					GVL_MASTER.stNestTable.qNestRotatePortA := FALSE;
					GVL_MASTER.stNestTable.qNestRotatePortB := FALSE;
					GVL_MASTER.stNestTable.bNestInMotion    := FALSE;
				
					GVL_MASTER.stProcess.bNestTestingReady  := FALSE;
					GVL_MASTER.stProcess.bReleaseNestRotation := FALSE;
				
					GVL_MASTER.stNestTable.bSupportExtendRequest  := FALSE;
					GVL_MASTER.stNestTable.bSupportRetractRequest := TRUE;
				
					GVL_MASTER.stMachineStatus.eMachineState := E_MachineState.FAULT;

        END_CASE

    // =================================================================
    // FAULT 
    // =================================================================
	
	E_MachineState.FAULT:
	
	 				GVL_MASTER.stNestTable.qNestRotatePortA := FALSE;
					GVL_MASTER.stNestTable.qNestRotatePortB := FALSE;
					GVL_MASTER.stNestTable.bNestInMotion    := FALSE;
				
					GVL_MASTER.stProcess.bNestTestingReady  := FALSE;
					GVL_MASTER.stProcess.bReleaseNestRotation := FALSE;
				
					GVL_MASTER.stNestTable.bSupportExtendRequest  := FALSE;
					GVL_MASTER.stNestTable.bSupportRetractRequest := TRUE;

	    IF GVL_IO.stSafety.bSafetyOK AND NOT GVL_Master.stMachineStatus.bFault THEN
        	eNestState := E_NestState.IDLE;
        END_IF

	

		
	END_CASE
END_METHOD

METHOD PRIVATE M_OperatorExchangeControl
VAR
	iOperatorNestIndex 	: INT;
    bOperatorResultPass : BOOL;
    bOperatorResultFail : BOOL;
	bOperatorResultValid : BOOL;
END_VAR
// ============================================================================
// MERGED OPERATOR EXCHANGE CONTROL
//
// Base:
//     - Immediate retention of one-scan removal and reject pulses.
//     - Complete enabled/disabled Puck Locker behavior.
//     - Recovery if the Puck Locker mode changes during an exchange.
//
// Merge adjustments:
//     - Permit a pending PASS or FAIL result to be handled while another nest
//       is in TESTING.
//     - Prevent WaitingForPartLoading from blocking when the locker is disabled.
// ============================================================================
// Default value prevents stale index permission.
bOperatorExchangeComplete := FALSE;


// -----------------------------------------------------------------------------
// Validate the nest currently accessible to the operator.
// -----------------------------------------------------------------------------
IF eOperatorNestPosition = E_NestPosition.Unknown THEN
    RETURN;
END_IF


iOperatorNestIndex := TO_INT(eOperatorNestPosition);

IF (iOperatorNestIndex < 1) OR (iOperatorNestIndex > 4) THEN
    RETURN;
END_IF


// -----------------------------------------------------------------------------
// Result associated with the nest currently accessible to the operator.
// -----------------------------------------------------------------------------
bOperatorResultValid :=
    GVL_MASTER.astNestProcessResult[
        iOperatorNestIndex
    ].bResultValid;


bOperatorResultPass :=
    GVL_MASTER.astNestProcessResult[
        iOperatorNestIndex
    ].bResultValid
    AND
    GVL_MASTER.astNestProcessResult[
        iOperatorNestIndex
    ].bPass;


bOperatorResultFail :=
    GVL_MASTER.astNestProcessResult[
        iOperatorNestIndex
    ].bResultValid
    AND
    GVL_MASTER.astNestProcessResult[
        iOperatorNestIndex
    ].bFail;

// -----------------------------------------------------------------------------
// Retain operator actions even while the Kistler is processing another nest.
//
// Both the nest removal pulse and the reject sensor pulse last only one PLC
// scan. They must therefore be retained immediately and not only when the
// exchange state machine reaches the corresponding waiting state.
// -----------------------------------------------------------------------------

// A processed part was removed from the operator nest.
IF (
        bOperatorResultValid
        OR bPendingOperatorResultPass
        OR bPendingOperatorResultFail
   )
   AND GVL_MASTER.astNestTracking[
        iOperatorNestIndex
   ].bPartRemovedPulse THEN

    bPartRemovedConfirmedForExchange := TRUE;

END_IF


// -----------------------------------------------------------------------------
// A new part was loaded into the operator nest.
//
// The previous part result may remain latched in the exchange state machine,
// but the newly loaded physical part has not yet been tested.
//
// Clear only the HMI measurement/result so the new part is displayed as NONE.
// -----------------------------------------------------------------------------
IF GVL_MASTER.astNestTracking[
        iOperatorNestIndex
   ].bPartLoadedPulse THEN

    // Preserve the disposition of the removed part before clearing
    // the visual result for the newly loaded part.
    IF bOperatorResultValid THEN

        bPendingOperatorResultPass :=
            bOperatorResultPass;

        bPendingOperatorResultFail :=
            bOperatorResultFail;

    END_IF

    // The newly loaded part has not been tested yet.
    // Display NONE without losing the pending disposition above.
    M_HMIKistlerResult(
        eNestPosition := eOperatorNestPosition,
        bPartOK       := FALSE,
        bPartNOK      := FALSE,
        rForce        := 0.0,
        rDistance     := 0.0,
        bResetValues  := TRUE
    );

END_IF


// Reject confirmation is only valid after the failed part
// has been removed from the operator nest.
//
// Required order:
// 1. Remove the failed part from the nest.
// 2. Place the failed part at the reject sensor.
// 3. Complete the operator exchange.
IF (
        bOperatorResultFail
        OR bPendingOperatorResultFail
   )
   AND bPartRemovedConfirmedForExchange
   AND rtPartPresentReject.Q THEN

    bRejectConfirmedForExchange := TRUE;

END_IF


// ============================================================================
// Operator exchange sequence
// ============================================================================
CASE eOperatorExchangeState OF


    // ========================================================================
    E_OperatorExchangeState.Idle:
    // ========================================================================

        bOperatorExchangeComplete := FALSE;

        // Preserve the physical nest associated with this exchange.
        eCompletedOperatorExchangeNest :=
            eOperatorNestPosition;


        // --------------------------------------------------------------------
        // Case 1:
        // A tested result is pending at the operator nest.
        //
        // The processed part must be handled before the table may index.
        // --------------------------------------------------------------------
        IF
			(
				(
					eNestState = E_NestState.IDLE
					OR
					eNestState = E_NestState.WAIT_OPERATOR_EXCHANGE
					OR
					eNestState = E_NestState.TESTING
				)
				AND NOT GVL_MASTER.stNestTable.bNestInMotion
				AND GVL_MASTER.stNestTable.bNestReadySensor
				AND GVL_MASTER.stNestTable.bNestLockedSensor
				AND bOperatorResultValid
			)
			THEN

            // Latch the result for the entire operator exchange.
            //
            // Do not reset these variables every PLC cycle.
            bPendingOperatorResultPass :=
                bOperatorResultPass;

            bPendingOperatorResultFail :=
                bOperatorResultFail;

           bRejectConfirmedForExchange := FALSE;


			// -------------------------------------------------------------
			// The processed part may already have been removed while another
			// nest was being tested.
			//
			// If the operator already loaded a new part, the physical sensor
			// will be ON again. Therefore, the retained removal event must
			// take priority over the current sensor state.
			// -------------------------------------------------------------
			IF bPartRemovedConfirmedForExchange THEN
			
				// ---------------------------------------------------------
				// PASS result.
				// ---------------------------------------------------------
				IF bOperatorResultPass THEN
			
					IF GVL_HMI.stPuckLocker.eMode =
						E_PuckLockerMode.Disabled THEN
			
						eOperatorExchangeState :=
							E_OperatorExchangeState.ExchangeComplete;
			
					ELSE
			
						eOperatorExchangeState :=
							E_OperatorExchangeState.WaitingForPuckRemoval;
			
					END_IF
			
			
				// ---------------------------------------------------------
				// FAIL result.
				// ---------------------------------------------------------
				ELSIF bOperatorResultFail THEN
			
					eOperatorExchangeState :=
						E_OperatorExchangeState.WaitingForRejectConfirmation;
			
				END_IF
			
			
			// -------------------------------------------------------------
			// No removal event was retained and the processed part is still
			// physically present.
			//
			// Wait for the operator to remove it.
			// -------------------------------------------------------------
			ELSIF GVL_MASTER.stSensors.bPartPresent_NEST THEN
			
				eOperatorExchangeState :=
					E_OperatorExchangeState.WaitingForPartRemoval;
			
			
			// -------------------------------------------------------------
			// The part is already absent, for example after fault recovery
			// or machine restart.
			// -------------------------------------------------------------
			ELSE
			


				bPartRemovedConfirmedForExchange := TRUE;
			
				// ---------------------------------------------------------
				// PASS result.
				// ---------------------------------------------------------
				IF bOperatorResultPass THEN
			
					IF GVL_HMI.stPuckLocker.eMode =
						E_PuckLockerMode.Disabled THEN
			
						eOperatorExchangeState :=
							E_OperatorExchangeState.ExchangeComplete;
			
					ELSE
			
						eOperatorExchangeState :=
							E_OperatorExchangeState.WaitingForPuckRemoval;
			
					END_IF
			
			
				// ---------------------------------------------------------
				// FAIL result.
				// ---------------------------------------------------------
			ELSIF bOperatorResultFail THEN
			
				// A valid FAIL result must always be physically confirmed
				// at the reject station before the exchange is completed.
				//
				// The part may already have been removed from the operator nest
				// before this state is evaluated, so the current part-present
				// sensor must not bypass reject confirmation.
				eOperatorExchangeState :=
					E_OperatorExchangeState.WaitingForRejectConfirmation;
			
			END_IF
			
			END_IF


        // --------------------------------------------------------------------
        // Case 2:
        // No tested result is pending.
        //
        // Enabled:
        //     Require a present and locked puck.
        //
        // Disabled:
        //     Ignore only the physical puck conditions.
        // --------------------------------------------------------------------
        ELSIF (
                eNestState = E_NestState.IDLE
                OR
                eNestState = E_NestState.WAIT_OPERATOR_EXCHANGE
              )
              AND NOT GVL_MASTER.stNestTable.bNestInMotion
              AND GVL_MASTER.stNestTable.bNestReadySensor
			  AND NOT bPendingOperatorResultPass
			  AND NOT bPendingOperatorResultFail
              AND GVL_MASTER.stNestTable.bNestLockedSensor
              AND NOT bOperatorResultValid
              AND (
                    GVL_HMI.stPuckLocker.eMode =
                        E_PuckLockerMode.Disabled

                    OR
                    (
                        GVL_MASTER.stPuckLocker.bPuckDetected
                        AND
                        GVL_MASTER.stPuckLocker.bPuckLocked
                        AND
                        GVL_MASTER.stPuckLocker.eState =
                            E_PuckLockerState.Locked
                    )
              ) THEN

            bPendingOperatorResultPass := FALSE;
            bPendingOperatorResultFail := FALSE;

            bPartRemovedConfirmedForExchange := FALSE;
            bRejectConfirmedForExchange := FALSE;

            eOperatorExchangeState :=
                E_OperatorExchangeState.ExchangeComplete;

        END_IF


    // ========================================================================
    E_OperatorExchangeState.WaitingForPartRemoval:
    // ========================================================================

        bOperatorExchangeComplete := FALSE;


        // This state is entered only when a processed part was confirmed
        // present in the operator nest.
        //
        // Therefore, the part has been removed when the physical sensor
        // becomes FALSE.
        IF bPartRemovedConfirmedForExchange
   			OR NOT GVL_MASTER.stSensors.bPartPresent_NEST THEN

            bPartRemovedConfirmedForExchange := TRUE;


            // -------------------------------------------------------------
            // PASS result.
            // -------------------------------------------------------------
            IF bPendingOperatorResultPass THEN

                // With the Puck Locker disabled, removal of the good part
                // completes the operator exchange.
                IF GVL_HMI.stPuckLocker.eMode =
                    E_PuckLockerMode.Disabled THEN

                    bPartRemovedConfirmedForExchange := FALSE;

                    eOperatorExchangeState :=
                        E_OperatorExchangeState.ExchangeComplete;

                ELSE

                    // Original enabled Puck Locker sequence.
                    eOperatorExchangeState :=
                        E_OperatorExchangeState.WaitingForPuckRemoval;

                END_IF


            // -------------------------------------------------------------
            // FAIL result.
            // -------------------------------------------------------------
            ELSIF bPendingOperatorResultFail THEN

                // The rejected part must be placed at the reject sensor.
                eOperatorExchangeState :=
                    E_OperatorExchangeState.WaitingForRejectConfirmation;

            END_IF

        END_IF


    // ========================================================================
    E_OperatorExchangeState.WaitingForPuckRemoval:
    // ========================================================================

        bOperatorExchangeComplete := FALSE;


        // Recovery protection:
        //
        // If the Puck Locker is disabled while the sequence is already in
        // this state, no puck removal must be awaited.
        IF GVL_HMI.stPuckLocker.eMode =
            E_PuckLockerMode.Disabled THEN

            bPartRemovedConfirmedForExchange := FALSE;

            eOperatorExchangeState :=
                E_OperatorExchangeState.ExchangeComplete;

        ELSE

            // Once the locker accepts the release request,
            // the part-removal handshake is no longer needed.
            IF GVL_MASTER.stPuckLocker.eState =
                E_PuckLockerState.ReleasingPuck THEN

                bPartRemovedConfirmedForExchange := FALSE;

            END_IF


            // Advance when the old puck is physically gone.
            //
            // Do not require the locker to remain in ReleasingPuck.
            IF NOT GVL_MASTER.stPuckLocker.bPuckDetected THEN

                eOperatorExchangeState :=
                    E_OperatorExchangeState.WaitingForNewPuck;

            END_IF

        END_IF


    // ========================================================================
    E_OperatorExchangeState.WaitingForRejectConfirmation:
    // ========================================================================

        bOperatorExchangeComplete := FALSE;


        // Latch the reject-bin sensor pulse.
        IF rtPartPresentReject.Q THEN

            bRejectConfirmedForExchange := TRUE;

        END_IF


        // Complete the rejected-part exchange when:
        //
        // 1. The rejected part has been confirmed at the reject sensor.
        // 2. The part is no longer present in the operator nest.
        // 3. The Puck Locker is disabled, or the puck remains present
        //    and locked.
        IF bRejectConfirmedForExchange
			   AND bPartRemovedConfirmedForExchange
			   AND
			   (
                GVL_HMI.stPuckLocker.eMode =
                    E_PuckLockerMode.Disabled

                OR
                (
                    GVL_MASTER.stPuckLocker.bPuckDetected
                    AND
                    GVL_MASTER.stPuckLocker.bPuckLocked
                    AND
                    GVL_MASTER.stPuckLocker.eState =
                        E_PuckLockerState.Locked
                )
           ) THEN

            bPartRemovedConfirmedForExchange := FALSE;

            eOperatorExchangeState :=
                E_OperatorExchangeState.ExchangeComplete;

        END_IF


    // ========================================================================
    E_OperatorExchangeState.WaitingForNewPuck:
    // ========================================================================


        bOperatorExchangeComplete := FALSE;


        // Recovery protection:
        //
        // A replacement puck is not required when the locker is disabled.
        IF GVL_HMI.stPuckLocker.eMode =
            E_PuckLockerMode.Disabled THEN

            eOperatorExchangeState :=
                E_OperatorExchangeState.ExchangeComplete;


        // Original enabled Puck Locker sequence.
        ELSIF GVL_MASTER.stPuckLocker.bPuckDetected THEN

            eOperatorExchangeState :=
                E_OperatorExchangeState.WaitingForPuckLocked;

        END_IF


    // ========================================================================
    E_OperatorExchangeState.WaitingForPuckLocked:
    // ========================================================================

        bOperatorExchangeComplete := FALSE;


        // Recovery protection:
        //
        // Physical puck locking is not required when the locker is disabled.
        IF GVL_HMI.stPuckLocker.eMode =
            E_PuckLockerMode.Disabled THEN

            eOperatorExchangeState :=
                E_OperatorExchangeState.ExchangeComplete;


        // Original enabled Puck Locker sequence.
        ELSIF GVL_MASTER.stPuckLocker.bPuckDetected
           AND GVL_MASTER.stPuckLocker.bPuckLocked
           AND GVL_MASTER.stPuckLocker.eState =
                E_PuckLockerState.Locked THEN

            // Loading a new part remains optional.
            eOperatorExchangeState :=
                E_OperatorExchangeState.ExchangeComplete;

        END_IF


    // ========================================================================
    E_OperatorExchangeState.WaitingForPartLoading:
    // ========================================================================

        bOperatorExchangeComplete := FALSE;


        // Recovery protection:
        //
        // If the Puck Locker is disabled while this legacy state is active,
        // physical puck conditions must no longer block the exchange.
        IF GVL_HMI.stPuckLocker.eMode =
            E_PuckLockerMode.Disabled THEN

            eOperatorExchangeState :=
                E_OperatorExchangeState.ExchangeComplete;


        // Original enabled Puck Locker behavior.
        //
        // Require an actual OFF -> ON transition from the operator nest
        // sensor. The puck must also be present and locked.
        ELSIF GVL_MASTER.astNestTracking[
                iOperatorNestIndex
              ].bPartLoadedPulse
              AND GVL_MASTER.stPuckLocker.bPuckDetected
              AND GVL_MASTER.stPuckLocker.bPuckLocked
              AND GVL_MASTER.stPuckLocker.eState =
                    E_PuckLockerState.Locked THEN

            eOperatorExchangeState := E_OperatorExchangeState.ExchangeComplete;

        END_IF


    // ========================================================================
    E_OperatorExchangeState.ExchangeComplete:
    // ========================================================================

        // Keep the index permission active until the table starts moving.
        bOperatorExchangeComplete := TRUE;


        // The previous result and its disposition are complete.
        M_ClearCompletedOperatorNestResult();


        IF GVL_MASTER.stNestTable.bNestInMotion THEN

            bPendingOperatorResultPass := FALSE;
            bPendingOperatorResultFail := FALSE;

            bPartRemovedConfirmedForExchange := FALSE;
            bRejectConfirmedForExchange := FALSE;

            eOperatorExchangeState :=  E_OperatorExchangeState.WaitingForTableIndexComplete;

        END_IF


    // ========================================================================
    E_OperatorExchangeState.WaitingForTableIndexComplete:
    // ========================================================================

        bOperatorExchangeComplete := TRUE;

        IF eNestState = E_NestState.TESTING
           AND NOT GVL_MASTER.stNestTable.bNestInMotion
           AND GVL_MASTER.stNestTable.bNestReadySensor
           AND GVL_MASTER.stNestTable.bNestLockedSensor
           AND eCurrentNestPos <> E_NestPosition.Unknown THEN

            bOperatorExchangeComplete := FALSE;

            bPendingOperatorResultPass := FALSE;
            bPendingOperatorResultFail := FALSE;

            bPartRemovedConfirmedForExchange := FALSE;
            bRejectConfirmedForExchange := FALSE;

            eOperatorExchangeState :=  E_OperatorExchangeState.Idle;

        END_IF


    // ========================================================================
    ELSE
    // ========================================================================

        bOperatorExchangeComplete := FALSE;

        bPendingOperatorResultPass := FALSE;
        bPendingOperatorResultFail := FALSE;

        bPartRemovedConfirmedForExchange := FALSE;
        bRejectConfirmedForExchange := FALSE;

        eOperatorExchangeState := E_OperatorExchangeState.Idle;

END_CASE

// -----------------------------------------------------------------------------
// Reject popup control.
//
// Show the popup as soon as a failed part arrives at the operator position.
// Keep it visible after the part is removed while reject confirmation is
// still pending.
//
// The popup closes automatically when the reject sensor is confirmed and
// the operator exchange leaves WaitingForRejectConfirmation.
// -----------------------------------------------------------------------------
GVL_HMI.bShowRejectPopup :=
    (
        (
            eOperatorExchangeState =
                E_OperatorExchangeState.WaitingForPartRemoval
        )
        AND bPendingOperatorResultFail
    )
    OR
    (
        eOperatorExchangeState =
            E_OperatorExchangeState.WaitingForRejectConfirmation
    );
END_METHOD

METHOD PRIVATE M_PreExecution : BOOL
VAR

END_VAR
// =================================================================================
// SYSTEM TIMERS
// =================================================================================
// Update initialization and safety timers on every PLC scan cycle
tonSys_Init(IN := GVL_MASTER.stMachineStatus.bInitialising);
tonSys_InitTimeout(IN := GVL_MASTER.stMachineStatus.bInitialising);

// TwinSAFE circuit stabilization timer (10 seconds)
tonSafety(IN := (GVL_MASTER.stMachineStatus.eMachineState = E_MachineState.SAFETY), PT := T#10S);

// 
//  fbStopTrigger(CLK := GVL_Master.i_bButtonStop);
//  bButtonStop := fbStopTrigger.Q;

// =================================================================================
// HMI MESSAGE CLEARING
// =================================================================================
// Clear old system messages if the machine is not actively in production
// Uses the proper ENUM namespace from your MASTER folder
IF GVL_MASTER.stMachineStatus.eMachineState <> E_MachineState.SYSTEM_AUTO_CYCLE THEN
    sMachineMessage := '';            
END_IF


// =================================================================================
// CRITICAL FAULT INTERLOCK (Watchdog)
// =================================================================================
// If Kistler hardware is NOT ready, force the state machine to FAULT immediately
// Exception: Do not override if the system is currently in SAFETY or POWER_UP
IF NOT GVL_MASTER.bKistlerSystemReady 
    AND GVL_MASTER.stMachineStatus.eMachineState <> E_MachineState.SAFETY 
    AND GVL_MASTER.stMachineStatus.eMachineState <> E_MachineState.SYSTEM_POWER_UP THEN
    
    GVL_MASTER.stMachineStatus.eMachineState := E_MachineState.FAULT;
END_IF


// =================================================================================
// START LEDs BUTTON OFF
// =================================================================================
eMode_LED_Start := E_LEDs_Mode.OFF;
eMode_LED_Reset := E_LEDs_Mode.OFF;

// =================================================================================
// METHOD EXECUTION FEEDBACK (Return True)
// =================================================================================
// Returning TRUE confirms the pre-execution routine completed successfully
M_PreExecution := TRUE;
END_METHOD

METHOD M_ProcessCycle : BOOL
VAR
    bControlledStopActive 			: BOOL;
    rTrigTwoHands : R_TRIG;

    bManualIndexerOnly       		: BOOL;
    bManualKistlerOnly       		: BOOL;
    bManualIndexerAndKistler 		: BOOL;
	

    bCurrentNestFaultRejectPending : BOOL;


END_VAR
// ============================================================================
// MERGED M_ProcessCycle
// Base: Renan + Thays
// Includes disabled-nest handling, empty-nest result clearing and
// eLastTestedNestPos update for skipped new positions.
// ============================================================================

// Process cycle is allowed during:
//
// 1. Automatic production.
// 2. Manual Mode when the Kistler or indexer manual function is enabled.
bProcessCycleAllowed :=
    (GVL_MASTER.stMachineStatus.eMachineState =
        E_MachineState.SYSTEM_AUTO_CYCLE)
    OR
    (GVL_MASTER.stMachineStatus.eMachineState =
        E_MachineState.MANUAL_MODE
     AND
        (GVL_HMI.i_bHMIKistlerManualEnable
         OR GVL_HMI.i_bHMIIndexerManualEnable));

bManualIndexerOnly :=
    GVL_HMI.i_bHMIIndexerManualEnable
    AND NOT GVL_HMI.i_bHMIKistlerManualEnable;

bManualKistlerOnly :=
    GVL_HMI.i_bHMIKistlerManualEnable
    AND NOT GVL_HMI.i_bHMIIndexerManualEnable;

bManualIndexerAndKistler :=
    GVL_HMI.i_bHMIIndexerManualEnable
    AND GVL_HMI.i_bHMIKistlerManualEnable;

// -----------------------------------------------------------------------------
// If process execution is not permitted, reset the temporary process states.
//
// Stored nest PASS/FAIL results must not be cleared by M_ResetProcessCycle.
// -----------------------------------------------------------------------------
IF NOT bProcessCycleAllowed THEN

    M_ResetProcessCycle();

    RETURN;

END_IF

// -----------------------------------------------------------------------------
// Common timers and edge detections.
// -----------------------------------------------------------------------------
rTrigTwoHands(
    CLK := GVL_IO.stSafety.bTwoHandsSafe
);

tTwoHandTargetTime :=
    REAL_TO_TIME(rHmiTwoHandPresetTime);

tTwoHandHoldTimer(
    IN := GVL_IO.stSafety.bTwoHandsSafe,
    PT := tTwoHandTargetTime
);

rtPartPresentReject(
    CLK := GVL_MASTER.stSensors.bPartPresent_Reject
);

// ============================================================================
// COMMON POSITION AND TRACKING UPDATE
//
// These methods are required in both Auto and Manual Mode.
// ============================================================================
eCurrentNestPos := M_GetCurrentPosition();

M_UpdateActiveNestPositions();

M_UpdateOperatorNestTracking();

// =====================================================
// CURRENT KISTLER NEST - PART MEMORY
// =====================================================
// Read the stored part presence for the physical nest
// currently positioned at the Kistler station.

bCurrentNestPartLoaded := FALSE;

CASE eCurrentNestPos OF

    E_NestPosition.Position_1:
        bCurrentNestPartLoaded :=
            GVL_MASTER.astNestTracking[1].bPartLoaded;

    E_NestPosition.Position_2:
        bCurrentNestPartLoaded :=
            GVL_MASTER.astNestTracking[2].bPartLoaded;

    E_NestPosition.Position_3:
        bCurrentNestPartLoaded :=
            GVL_MASTER.astNestTracking[3].bPartLoaded;

    E_NestPosition.Position_4:
        bCurrentNestPartLoaded :=
            GVL_MASTER.astNestTracking[4].bPartLoaded;

ELSE
    bCurrentNestPartLoaded := FALSE;

END_CASE

// -----------------------------------------------------------------------------
// Determine safely whether the nest currently at the Kistler still contains
// a valid FAIL result.
//
// The enum is mapped explicitly to indexes 1..4 to prevent an invalid array
// access when the current position is UNKNOWN.
// -----------------------------------------------------------------------------
bCurrentNestFaultRejectPending := FALSE;

CASE eCurrentNestPos OF

    E_NestPosition.Position_1:

        bCurrentNestFaultRejectPending :=
            GVL_MASTER.astNestProcessResult[1].bResultValid
            AND GVL_MASTER.astNestProcessResult[1].bFail;

    E_NestPosition.Position_2:

        bCurrentNestFaultRejectPending :=
            GVL_MASTER.astNestProcessResult[2].bResultValid
            AND GVL_MASTER.astNestProcessResult[2].bFail;

    E_NestPosition.Position_3:

        bCurrentNestFaultRejectPending :=
            GVL_MASTER.astNestProcessResult[3].bResultValid
            AND GVL_MASTER.astNestProcessResult[3].bFail;

    E_NestPosition.Position_4:

        bCurrentNestFaultRejectPending :=
            GVL_MASTER.astNestProcessResult[4].bResultValid
            AND GVL_MASTER.astNestProcessResult[4].bFail;

ELSE

    bCurrentNestFaultRejectPending := FALSE;

END_CASE

// ============================================================================
// AUTOMATIC OPERATOR EXCHANGE
//
// The following methods belong only to automatic production.
//
// They must not:
//
// - send a PASS/FAIL disposition while in Manual Mode;
// - release a puck during Manual Mode;
// - clear a completed nest result during Manual Mode;
// - block manual index movement waiting for part removal;
// - block manual index movement waiting for reject confirmation;
// - block manual index movement waiting for a puck.
// ============================================================================
IF GVL_MASTER.stMachineStatus.eMachineState =
    E_MachineState.SYSTEM_AUTO_CYCLE THEN

    M_UpdatePuckLockerPartRemovalStatus();

    M_ConfirmPuckLockerDisposition();

    M_PuckLockerDisposition();

    M_OperatorExchangeControl();

ELSE

    // Prevent a stale removal confirmation from being sent to the
    // Puck Locker while the machine is operating manually.
    GVL_MASTER.stPuckLocker.bPartRemovedFromNest := FALSE;

END_IF

// -----------------------------------------------------------------------------
// Determine whether the current physical table position is different from
// the most recently processed Kistler position.
// -----------------------------------------------------------------------------
bNestNewPositionReady :=
    (
        eCurrentNestPos <> E_NestPosition.UNKNOWN
    )
    AND
    (
        eCurrentNestPos <> eLastTestedNestPos
    );







// -----------------------------------------------------------------------------
// Capture maximum Kistler distance during Auto Cycle.
//
// The Kistler position returns to zero after the test, therefore only a
// distance greater than the value already stored is accepted.
// -----------------------------------------------------------------------------
IF GVL_MASTER.stProcess.bKistlerCycleRequest
   AND NOT stKistlerOutTelegram.bSequenceEnd
   AND GVL_MASTER.stMachineStatus.eMachineState =
       E_MachineState.SYSTEM_AUTO_CYCLE THEN

    CASE eCurrentNestPos OF

        E_NestPosition.Position_1:

            IF stKistler_Status.rLiveDistance >
               GVL_HMI.aKistlerNestResult[1].rDistance THEN

                GVL_HMI.aKistlerNestResult[1].rDistance :=
                    stKistler_Status.rLiveDistance;

            END_IF


        E_NestPosition.Position_2:

            IF stKistler_Status.rLiveDistance >
               GVL_HMI.aKistlerNestResult[2].rDistance THEN

                GVL_HMI.aKistlerNestResult[2].rDistance :=
                    stKistler_Status.rLiveDistance;

            END_IF


        E_NestPosition.Position_3:

            IF stKistler_Status.rLiveDistance >
               GVL_HMI.aKistlerNestResult[3].rDistance THEN

                GVL_HMI.aKistlerNestResult[3].rDistance :=
                    stKistler_Status.rLiveDistance;

            END_IF


        E_NestPosition.Position_4:

            IF stKistler_Status.rLiveDistance >
               GVL_HMI.aKistlerNestResult[4].rDistance THEN

                GVL_HMI.aKistlerNestResult[4].rDistance :=
                    stKistler_Status.rLiveDistance;

            END_IF

    END_CASE

END_IF

// -----------------------------------------------------------------------------
// Capture live Kistler values while an automatic or manual sequence is active.
//
// This does not store PASS/FAIL. It only updates the live maximum values.
// -----------------------------------------------------------------------------
// -----------------------------------------------------------------------------
// Capture live Kistler values during Manual Mode only.
//
// Automatic production results must not be updated while the Kistler sequence
// is still running. AutoCycle stores the final measurement only after the
// Kistler sequence has completed.
// -----------------------------------------------------------------------------
IF GVL_MASTER.stProcess.bKistlerCycleRequest
   AND NOT stKistlerOutTelegram.bSequenceEnd
   AND GVL_MASTER.stMachineStatus.eMachineState =
       E_MachineState.MANUAL_MODE THEN

    CASE eCurrentNestPos OF

        E_NestPosition.Position_1:

            GVL_HMI.aKistlerManualResult[1].rForce :=
                uKistlerCurveYMax.rValue;

            IF stKistler_Status.rLiveDistance >
               GVL_HMI.aKistlerManualResult[1].rDistance THEN

                GVL_HMI.aKistlerManualResult[1].rDistance :=
                    stKistler_Status.rLiveDistance;

            END_IF


        E_NestPosition.Position_2:

            GVL_HMI.aKistlerManualResult[2].rForce :=
                uKistlerCurveYMax.rValue;

            IF stKistler_Status.rLiveDistance >
               GVL_HMI.aKistlerManualResult[2].rDistance THEN

                GVL_HMI.aKistlerManualResult[2].rDistance :=
                    stKistler_Status.rLiveDistance;

            END_IF


        E_NestPosition.Position_3:

            GVL_HMI.aKistlerManualResult[3].rForce :=
                uKistlerCurveYMax.rValue;

            IF stKistler_Status.rLiveDistance >
               GVL_HMI.aKistlerManualResult[3].rDistance THEN

                GVL_HMI.aKistlerManualResult[3].rDistance :=
                    stKistler_Status.rLiveDistance;

            END_IF


        E_NestPosition.Position_4:

            GVL_HMI.aKistlerManualResult[4].rForce :=
                uKistlerCurveYMax.rValue;

            IF stKistler_Status.rLiveDistance >
               GVL_HMI.aKistlerManualResult[4].rDistance THEN

                GVL_HMI.aKistlerManualResult[4].rDistance :=
                    stKistler_Status.rLiveDistance;

            END_IF

    END_CASE

END_IF

// ============================================================================
// PROCESS CYCLE COORDINATOR
// ============================================================================
CASE GVL_MASTER.stMachineStatus.eMachineState OF

    // ========================================================================
    // AUTOMATIC CYCLE
    // ========================================================================
    E_MachineState.SYSTEM_AUTO_CYCLE:

        CASE eProcessCycleState OF

            // =================================================================
            E_ProcessCycle_State.IDLE:
            // =================================================================

                GVL_MASTER.stProcess.bKistlerCycleRequest := FALSE;
                GVL_MASTER.stProcess.bKistlerCycleDone    := FALSE;
                GVL_MASTER.stProcess.bKistlerHomeDone     := FALSE;
                GVL_MASTER.stProcess.bReleaseNestRotation := FALSE;

                tonAfterKistlerDelay(IN := FALSE);

                IF bProcessCycleAllowed THEN

                    eProcessCycleState :=
                        E_ProcessCycle_State.WAIT_NEST_TESTING_READY;

                END_IF

            // =================================================================
            E_ProcessCycle_State.WAIT_NEST_TESTING_READY:
            // =================================================================

                GVL_MASTER.stProcess.bKistlerCycleRequest := FALSE;
                GVL_MASTER.stProcess.bReleaseNestRotation := FALSE;

                tonAfterKistlerDelay(IN := FALSE);

                IF NOT bProcessCycleAllowed THEN

                    eProcessCycleState :=
                        E_ProcessCycle_State.IDLE;

                // -------------------------------------------------------------
                // Invalid table position.
                //
                // Never execute the Kistler if the PLC cannot determine which
                // physical nest is currently at the test station.
                // -------------------------------------------------------------
                ELSIF GVL_MASTER.stProcess.bNestTestingReady
                      AND eNestState = E_NestState.TESTING
                      AND eCurrentNestPos =
                            E_NestPosition.UNKNOWN THEN

                    GVL_MASTER.stProcess.bKistlerCycleRequest := FALSE;
                    GVL_MASTER.stProcess.bReleaseNestRotation := FALSE;
                    GVL_MASTER.stProcess.bKistlerCycleDone    := FALSE;
                    GVL_MASTER.stProcess.bKistlerHomeDone     := FALSE;

                    eProcessCycleState :=
                        E_ProcessCycle_State.FAULT;

                // -------------------------------------------------------------
                // Fault-recovery reject.
                // -------------------------------------------------------------
                ELSIF bFaultRejectActive
                      AND bCurrentNestFaultRejectPending
                      AND GVL_MASTER.stProcess.bNestTestingReady
                      AND eNestState = E_NestState.TESTING
                      AND GVL_MASTER.stNestTable.bNestReadySensor
                      AND GVL_MASTER.stNestTable.bNestLockedSensor
                      AND NOT GVL_MASTER.stNestTable.bNestInMotion
                      AND eCurrentNestPos <>
                            E_NestPosition.UNKNOWN THEN

                    GVL_MASTER.stProcess.bKistlerCycleRequest := FALSE;
                    GVL_MASTER.stProcess.bKistlerCycleDone    := FALSE;
                    GVL_MASTER.stProcess.bKistlerHomeDone     := TRUE;

                    GVL_MASTER.stProcess.bReleaseNestRotation :=
                        TRUE;

                    eProcessCycleState :=
                        E_ProcessCycle_State.RELEASE_NEST;

                // -------------------------------------------------------------
                // Same position already processed, or no part at Kistler.
                // -------------------------------------------------------------
                ELSIF GVL_MASTER.stProcess.bNestTestingReady
                      AND eNestState = E_NestState.TESTING
                      AND GVL_MASTER.stNestTable.bNestReadySensor
                      AND GVL_MASTER.stNestTable.bNestLockedSensor
                      AND NOT GVL_MASTER.stNestTable.bNestInMotion
                      AND eCurrentNestPos <>
                            E_NestPosition.UNKNOWN
                      AND
                      (
                          NOT bNestNewPositionReady
                          OR NOT GVL_MASTER.stSensors.bPartPresent_Kistler
						  OR NOT bCurrentNestPartLoaded
                      ) THEN

                    GVL_MASTER.stProcess.bKistlerCycleRequest := FALSE;
                    GVL_MASTER.stProcess.bKistlerCycleDone    := FALSE;

                    GVL_MASTER.stProcess.bKistlerHomeDone :=
                        TRUE;

                    IF bNestNewPositionReady THEN

                        M_HMIKistlerResult(
                            eNestPosition := eCurrentNestPos,
                            bPartOK       := FALSE,
                            bPartNOK      := FALSE,
                            rForce        := 0.0,
                            rDistance     := 0.0,
                            bResetValues  := TRUE
                        );

                        eLastTestedNestPos :=
                            eCurrentNestPos;

                    END_IF

                    GVL_MASTER.stProcess.bReleaseNestRotation :=
                        TRUE;

                    eProcessCycleState :=
                        E_ProcessCycle_State.RELEASE_NEST;

                // -------------------------------------------------------------
                // New enabled nest containing a part.
                //
                // Execute the Kistler sequence.
                // -------------------------------------------------------------
                ELSIF GVL_MASTER.stProcess.bNestTestingReady
                      AND eNestState = E_NestState.TESTING
                      AND GVL_MASTER.stNestTable.bNestReadySensor
                      AND GVL_MASTER.stNestTable.bNestLockedSensor
                      AND NOT GVL_MASTER.stNestTable.bNestInMotion
                      AND stKistler_Status.eKistlerState =
                            E_KistlerState.READY
                      AND NOT stKistler_Status.bError
                      AND NOT bKistlerRecoveryHomeRequest
                      AND bNestNewPositionReady
                      AND GVL_MASTER.stSensors.bPartPresent_Kistler
					  AND bCurrentNestPartLoaded
                      AND M_IsNestEnabled(eCurrentNestPos) THEN

                    GVL_MASTER.stProcess.bKistlerCycleDone := FALSE;
                    GVL_MASTER.stProcess.bKistlerHomeDone  := FALSE;

                    // A new automatic Kistler result has not yet been stored.
                    bKistlerResultStored := FALSE;

                    M_HMIKistlerResult(
                        eNestPosition := eCurrentNestPos,
                        bPartOK       := FALSE,
                        bPartNOK      := FALSE,
                        rForce        := 0.0,
                        rDistance     := 0.0,
                        bResetValues  := TRUE
                    );

                    eProcessCycleState :=
                        E_ProcessCycle_State.REQUEST_KISTLER;

                // -------------------------------------------------------------
                // Nest disabled from HMI.
                // -------------------------------------------------------------
                ELSIF GVL_MASTER.stProcess.bNestTestingReady
                      AND eNestState = E_NestState.TESTING
                      AND GVL_MASTER.stNestTable.bNestReadySensor
                      AND GVL_MASTER.stNestTable.bNestLockedSensor
                      AND NOT GVL_MASTER.stNestTable.bNestInMotion
                      AND eCurrentNestPos <>
                            E_NestPosition.UNKNOWN
                      AND bNestNewPositionReady
                      AND GVL_MASTER.stSensors.bPartPresent_Kistler
                      AND NOT M_IsNestEnabled(eCurrentNestPos) THEN

                    GVL_MASTER.stProcess.bKistlerCycleRequest := FALSE;
                    GVL_MASTER.stProcess.bKistlerCycleDone    := FALSE;
                    GVL_MASTER.stProcess.bKistlerHomeDone     := TRUE;

                    M_HMIKistlerResult(
                        eNestPosition := eCurrentNestPos,
                        bPartOK       := FALSE,
                        bPartNOK      := FALSE,
                        rForce        := 0.0,
                        rDistance     := 0.0,
                        bResetValues  := TRUE
                    );

                    eLastTestedNestPos :=
                        eCurrentNestPos;

                    GVL_MASTER.stProcess.bReleaseNestRotation :=
                        TRUE;

                    eProcessCycleState :=
                        E_ProcessCycle_State.RELEASE_NEST;

                END_IF

            // =================================================================
            E_ProcessCycle_State.REQUEST_KISTLER:
            // =================================================================

                GVL_MASTER.stProcess.bKistlerCycleRequest := TRUE;

                IF stKistler_Status.bError THEN

                    GVL_MASTER.stProcess.bKistlerCycleRequest :=
                        FALSE;

                    eProcessCycleState :=
                        E_ProcessCycle_State.FAULT;

                ELSIF stKistler_Status.eKistlerState <>
                      E_KistlerState.READY THEN

                    eProcessCycleState :=
                        E_ProcessCycle_State.WAIT_KISTLER_DONE;

                END_IF

            // =================================================================
            E_ProcessCycle_State.WAIT_KISTLER_DONE:
            // =================================================================

                GVL_MASTER.stProcess.bKistlerCycleRequest := TRUE;

                IF stKistler_Status.bError THEN

                    GVL_MASTER.stProcess.bKistlerCycleRequest :=
                        FALSE;

                    eProcessCycleState :=
                        E_ProcessCycle_State.FAULT;

                ELSIF stKistler_Status.eKistlerState =
                      E_KistlerState.DONE THEN

                    GVL_MASTER.stProcess.bKistlerCycleRequest :=
                        FALSE;

                    GVL_MASTER.stProcess.bKistlerCycleDone :=
                        TRUE;

                    eProcessCycleState :=
                        E_ProcessCycle_State.WAIT_KISTLER_HOME;

                END_IF

            // =================================================================
            E_ProcessCycle_State.WAIT_KISTLER_HOME:
            // =================================================================

                M_StoreKistlerResult();

                GVL_MASTER.stProcess.bKistlerCycleRequest := FALSE;

                IF stKistler_Status.bError THEN

                    eProcessCycleState :=
                        E_ProcessCycle_State.FAULT;

                ELSIF stKistlerOutTelegram.bHomePosReached
                      OR stKistlerOutTelegram.bRefPosReached
                      OR stKistler_Status.bInPosition THEN

                    GVL_MASTER.test :=
                        GVL_MASTER.test + 1;

                    GVL_MASTER.stProcess.bKistlerHomeDone :=
                        TRUE;

                    GVL_MASTER.stProcess.bKistlerCycleDone :=
                        TRUE;

                    // ---------------------------------------------------------
                    // Store the process result.
                    // ---------------------------------------------------------
                    IF stKistler_Status.bPartOK THEN

                        GVL_MASTER.stProcess.bKistlerResultOK :=
                            TRUE;

                        GVL_MASTER.stProcess.bKistlerResultNOK :=
                            FALSE;

                    ELSIF stKistler_Status.bPartNOK THEN

                        GVL_MASTER.stProcess.bKistlerResultOK :=
                            FALSE;

                        GVL_MASTER.stProcess.bKistlerResultNOK :=
                            TRUE;

                    ELSE

                        // Test ended without a valid OK/NOK result.
                        // Preserve the existing behavior.
                        RETURN;

                    END_IF

                    eLastTestedNestPos :=
                        eCurrentNestPos;

                    // ---------------------------------------------------------
                    // Store the final Kistler values for this nest.
                    //
                    // The result is stored only after the Kistler sequence has
                    // completed and Home / Ref / InPosition is confirmed.
                    // ---------------------------------------------------------
                    IF NOT M_HMIKistlerResult(
                        eNestPosition := eCurrentNestPos,
                        bPartOK       := stKistler_Status.bPartOK,
                        bPartNOK      := stKistler_Status.bPartNOK,
                        rForce        := uKistlerCurveYMax.rValue,
                        rDistance     := stKistler_Status.rLiveDistance,
                        bResetValues  := FALSE
                    ) THEN

                        RETURN;

                    END_IF

                    // ---------------------------------------------------------
                    // The final automatic result is now available.
                    //
                    // Statistics / Data History / CSV must only consume the
                    // result after this point.
                    // ---------------------------------------------------------
                    bKistlerResultStored := TRUE;

                    eProcessCycleState :=
                        E_ProcessCycle_State.WAIT_AFTER_KISTLER;

                END_IF

            // =================================================================
            E_ProcessCycle_State.WAIT_AFTER_KISTLER:
            // =================================================================

                IF stKistlerOutTelegram.bSequenceEnd
                   AND
                   (
                       stKistlerOutTelegram.bHomePosReached
                       OR
                       stKistlerOutTelegram.bRefPosReached
                       OR
                       stKistler_Status.bInPosition
                   ) THEN

                    GVL_MASTER.stProcess.bReleaseNestRotation :=
                        TRUE;

                    eProcessCycleState :=
                        E_ProcessCycle_State.RELEASE_NEST;

                END_IF

            // =================================================================
            E_ProcessCycle_State.RELEASE_NEST:
            // =================================================================

                GVL_MASTER.stProcess.bReleaseNestRotation := TRUE;

                IF eNestState <> E_NestState.TESTING
                   OR NOT GVL_MASTER.stProcess.bNestTestingReady THEN

                    GVL_MASTER.stProcess.bReleaseNestRotation :=
                        FALSE;

                    GVL_MASTER.stProcess.bKistlerCycleRequest :=
                        FALSE;

                    GVL_MASTER.stProcess.bKistlerCycleDone :=
                        FALSE;

                    GVL_MASTER.stProcess.bKistlerHomeDone :=
                        FALSE;

                    tonAfterKistlerDelay(IN := FALSE);

                    eProcessCycleState :=
                        E_ProcessCycle_State.WAIT_NEST_TESTING_READY;

                END_IF

            // =================================================================
            E_ProcessCycle_State.FAULT:
            // =================================================================

                GVL_MASTER.stProcess.bKistlerCycleRequest := FALSE;
                GVL_MASTER.stProcess.bReleaseNestRotation := FALSE;

                tonAfterKistlerDelay(IN := FALSE);

                M_ResetProcessCycle();

                GVL_MASTER.stMachineStatus.eMachineState :=
                    E_MachineState.FAULT;

                IF GVL_MASTER.stMachineStatus.bStopped THEN

                    eProcessCycleState :=
                        E_ProcessCycle_State.IDLE;

                END_IF

            // =================================================================
            ELSE
            // =================================================================

                eProcessCycleState :=
                    E_ProcessCycle_State.IDLE;

        END_CASE

    // ========================================================================
    // MANUAL MODE
    // ========================================================================
    E_MachineState.MANUAL_MODE:

        CASE eProcessCycleState OF

            // =================================================================
            E_ProcessCycle_State.IDLE:
            // =================================================================

                GVL_MASTER.stProcess.bKistlerCycleRequest := FALSE;
                GVL_MASTER.stProcess.bKistlerCycleDone := FALSE;
                GVL_MASTER.stProcess.bKistlerHomeDone := FALSE;
                GVL_MASTER.stProcess.bReleaseNestRotation := FALSE;

                GVL_MASTER.stProcess.bKistlerResultOK := FALSE;
                GVL_MASTER.stProcess.bKistlerResultNOK := FALSE;

                tonAfterKistlerDelay(IN := FALSE);

                // -------------------------------------------------------------
                // Manual indexer only or indexer + Kistler.
                // Wait until the table reaches the testing position.
                // -------------------------------------------------------------
                IF bManualIndexerOnly
                   OR bManualIndexerAndKistler THEN

                    eProcessCycleState :=
                        E_ProcessCycle_State.WAIT_NEST_TESTING_READY;

                // -------------------------------------------------------------
                // Manual Kistler only.
                // Prepare a new test and wait for the two-hand rising edge.
                // -------------------------------------------------------------
                ELSIF bManualKistlerOnly
                      AND NOT GVL_MASTER.stProcess.bNestTestingReady
                      AND stKistler_Status.eKistlerState =
                            E_KistlerState.READY
                      AND NOT stKistler_Status.bError
                      AND NOT bKistlerRecoveryHomeRequest THEN

                    GVL_MASTER.stProcess.bNestTestingReady := FALSE;

                    bKistlerResultStored := FALSE;
                    rKistlerCycleMaxForce := 0.0;
                    rKistlerCycleMaxDistance := 0.0;

                    CASE eCurrentNestPos OF

                        E_NestPosition.Position_1:
                            GVL_HMI.aKistlerManualResult[1].eResult :=
                                E_HMIKistlerResult.NONE;
                            GVL_HMI.aKistlerManualResult[1].rForce := 0.0;
                            GVL_HMI.aKistlerManualResult[1].rDistance := 0.0;

                        E_NestPosition.Position_2:
                            GVL_HMI.aKistlerManualResult[2].eResult :=
                                E_HMIKistlerResult.NONE;
                            GVL_HMI.aKistlerManualResult[2].rForce := 0.0;
                            GVL_HMI.aKistlerManualResult[2].rDistance := 0.0;

                        E_NestPosition.Position_3:
                            GVL_HMI.aKistlerManualResult[3].eResult :=
                                E_HMIKistlerResult.NONE;
                            GVL_HMI.aKistlerManualResult[3].rForce := 0.0;
                            GVL_HMI.aKistlerManualResult[3].rDistance := 0.0;

                        E_NestPosition.Position_4:
                            GVL_HMI.aKistlerManualResult[4].eResult :=
                                E_HMIKistlerResult.NONE;
                            GVL_HMI.aKistlerManualResult[4].rForce := 0.0;
                            GVL_HMI.aKistlerManualResult[4].rDistance := 0.0;

                    END_CASE

                    eProcessCycleState :=
                        E_ProcessCycle_State.REQUEST_KISTLER;

                END_IF

            // =================================================================
            E_ProcessCycle_State.WAIT_NEST_TESTING_READY:
            // =================================================================

                GVL_MASTER.stProcess.bKistlerCycleRequest := FALSE;
                GVL_MASTER.stProcess.bReleaseNestRotation := FALSE;

                tonAfterKistlerDelay(IN := FALSE);

                IF NOT (
                    bManualIndexerOnly
                    OR bManualIndexerAndKistler
                ) THEN

                    eProcessCycleState :=
                        E_ProcessCycle_State.IDLE;

                ELSIF GVL_MASTER.stProcess.bNestTestingReady
                      AND eNestState = E_NestState.TESTING
                      AND bManualIndexerAndKistler
                      AND stKistler_Status.eKistlerState =
                            E_KistlerState.READY
                      AND NOT stKistler_Status.bError
                      AND NOT bKistlerRecoveryHomeRequest
                      AND eCurrentNestPos <>
                            E_NestPosition.UNKNOWN THEN

                    GVL_MASTER.stProcess.bKistlerCycleDone := FALSE;
                    GVL_MASTER.stProcess.bKistlerHomeDone := FALSE;

                    bKistlerResultStored := FALSE;
                    rKistlerCycleMaxForce := 0.0;
                    rKistlerCycleMaxDistance := 0.0;

                    CASE eCurrentNestPos OF

                        E_NestPosition.Position_1:
                            GVL_HMI.aKistlerManualResult[1].eResult :=
                                E_HMIKistlerResult.NONE;
                            GVL_HMI.aKistlerManualResult[1].rForce := 0.0;
                            GVL_HMI.aKistlerManualResult[1].rDistance := 0.0;

                        E_NestPosition.Position_2:
                            GVL_HMI.aKistlerManualResult[2].eResult :=
                                E_HMIKistlerResult.NONE;
                            GVL_HMI.aKistlerManualResult[2].rForce := 0.0;
                            GVL_HMI.aKistlerManualResult[2].rDistance := 0.0;

                        E_NestPosition.Position_3:
                            GVL_HMI.aKistlerManualResult[3].eResult :=
                                E_HMIKistlerResult.NONE;
                            GVL_HMI.aKistlerManualResult[3].rForce := 0.0;
                            GVL_HMI.aKistlerManualResult[3].rDistance := 0.0;

                        E_NestPosition.Position_4:
                            GVL_HMI.aKistlerManualResult[4].eResult :=
                                E_HMIKistlerResult.NONE;
                            GVL_HMI.aKistlerManualResult[4].rForce := 0.0;
                            GVL_HMI.aKistlerManualResult[4].rDistance := 0.0;

                    END_CASE

                    eProcessCycleState :=
                        E_ProcessCycle_State.REQUEST_KISTLER;

                // -------------------------------------------------------------
                // Manual indexer only.
                // -------------------------------------------------------------
                ELSIF GVL_MASTER.stProcess.bNestTestingReady
                      AND eNestState = E_NestState.TESTING
                      AND bManualIndexerOnly THEN

                    GVL_MASTER.stProcess.bKistlerCycleRequest := FALSE;
                    GVL_MASTER.stProcess.bKistlerHomeDone := TRUE;
                    GVL_MASTER.stProcess.bReleaseNestRotation := TRUE;

                    eProcessCycleState :=
                        E_ProcessCycle_State.RELEASE_NEST;

                END_IF

            // =================================================================
            E_ProcessCycle_State.REQUEST_KISTLER:
            // =================================================================

                IF stKistler_Status.eKistlerState <>
                    E_KistlerState.READY THEN

                    eProcessCycleState :=
                        E_ProcessCycle_State.WAIT_KISTLER_DONE;

                ELSIF bManualKistlerOnly
                      AND GVL_IO.stSafety.bSafetyOK
                      AND rTrigTwoHands.Q
                      AND GVL_MASTER.stNestTable.bNestReadySensor
                      AND GVL_MASTER.stNestTable.bNestLockedSensor
                      AND NOT stKistler_Status.bError
                      AND NOT bKistlerRecoveryHomeRequest THEN

                    GVL_MASTER.stProcess.bKistlerCycleRequest := TRUE;

                ELSIF bManualIndexerAndKistler
                      AND GVL_MASTER.stProcess.bNestTestingReady
                      AND eNestState = E_NestState.TESTING
                      AND GVL_MASTER.stNestTable.bNestReadySensor
                      AND GVL_MASTER.stNestTable.bNestLockedSensor
                      AND NOT GVL_MASTER.stNestTable.bNestInMotion
                      AND eCurrentNestPos <>
                            E_NestPosition.UNKNOWN
                      AND bNestNewPositionReady
                      AND NOT stKistler_Status.bError
                      AND NOT bKistlerRecoveryHomeRequest THEN

                    GVL_MASTER.stProcess.bKistlerCycleRequest := TRUE;

                ELSIF stKistler_Status.bError THEN

                    GVL_MASTER.stProcess.bKistlerCycleRequest := FALSE;

                    eProcessCycleState :=
                        E_ProcessCycle_State.FAULT;

                END_IF

            // =================================================================
			E_ProcessCycle_State.WAIT_KISTLER_DONE:
			// =================================================================
			
				GVL_MASTER.stProcess.bKistlerCycleRequest := TRUE;
			
				IF stKistler_Status.bError THEN
			
					GVL_MASTER.stProcess.bKistlerCycleRequest := FALSE;
			
					eProcessCycleState :=
						E_ProcessCycle_State.FAULT;
			
				ELSIF stKistler_Status.eKistlerState =
					  E_KistlerState.DONE THEN
			
					GVL_MASTER.stProcess.bKistlerCycleRequest := FALSE;
					GVL_MASTER.stProcess.bKistlerCycleDone := TRUE;
			
					// Finalize the Kistler result.
					M_StoreKistlerResult();
			
					CASE eCurrentNestPos OF
			
						E_NestPosition.Position_1:
			
							GVL_HMI.aKistlerManualResult[1].rForce :=
								uKistlerCurveYMax.rValue;
			
							IF stKistler_Status.bPartOK THEN
								GVL_HMI.aKistlerManualResult[1].eResult :=
									E_HMIKistlerResult.PASS;
							ELSIF stKistler_Status.bPartNOK THEN
								GVL_HMI.aKistlerManualResult[1].eResult :=
									E_HMIKistlerResult.FAIL;
							ELSE
								GVL_HMI.aKistlerManualResult[1].eResult :=
									E_HMIKistlerResult.NONE;
							END_IF
			
			
						E_NestPosition.Position_2:
			
							GVL_HMI.aKistlerManualResult[2].rForce :=
								uKistlerCurveYMax.rValue;
			
							IF stKistler_Status.bPartOK THEN
								GVL_HMI.aKistlerManualResult[2].eResult :=
									E_HMIKistlerResult.PASS;
							ELSIF stKistler_Status.bPartNOK THEN
								GVL_HMI.aKistlerManualResult[2].eResult :=
									E_HMIKistlerResult.FAIL;
							ELSE
								GVL_HMI.aKistlerManualResult[2].eResult :=
									E_HMIKistlerResult.NONE;
							END_IF
			
			
						E_NestPosition.Position_3:
			
							GVL_HMI.aKistlerManualResult[3].rForce :=
								uKistlerCurveYMax.rValue;
			
							IF stKistler_Status.bPartOK THEN
								GVL_HMI.aKistlerManualResult[3].eResult :=
									E_HMIKistlerResult.PASS;
							ELSIF stKistler_Status.bPartNOK THEN
								GVL_HMI.aKistlerManualResult[3].eResult :=
									E_HMIKistlerResult.FAIL;
							ELSE
								GVL_HMI.aKistlerManualResult[3].eResult :=
									E_HMIKistlerResult.NONE;
							END_IF
			
			
						E_NestPosition.Position_4:
			
							GVL_HMI.aKistlerManualResult[4].rForce :=
								uKistlerCurveYMax.rValue;
			
							IF stKistler_Status.bPartOK THEN
								GVL_HMI.aKistlerManualResult[4].eResult :=
									E_HMIKistlerResult.PASS;
							ELSIF stKistler_Status.bPartNOK THEN
								GVL_HMI.aKistlerManualResult[4].eResult :=
									E_HMIKistlerResult.FAIL;
							ELSE
								GVL_HMI.aKistlerManualResult[4].eResult :=
									E_HMIKistlerResult.NONE;
							END_IF
			
					END_CASE
			
					IF bManualIndexerAndKistler THEN
			
						eLastTestedNestPos := eCurrentNestPos;
			
						eProcessCycleState :=
							E_ProcessCycle_State.WAIT_KISTLER_HOME;
			
					ELSE
			
						eProcessCycleState :=
							E_ProcessCycle_State.IDLE;
			
					END_IF
			
				END_IF

            // =================================================================
            E_ProcessCycle_State.WAIT_KISTLER_HOME:
            // =================================================================

                GVL_MASTER.stProcess.bKistlerCycleRequest := FALSE;

                IF stKistler_Status.bError THEN

                    eProcessCycleState :=
                        E_ProcessCycle_State.FAULT;

                ELSIF stKistlerOutTelegram.bHomePosReached
                      OR stKistlerOutTelegram.bRefPosReached
                      OR stKistler_Status.bInPosition THEN

                    GVL_MASTER.stProcess.bKistlerHomeDone := TRUE;

                    IF bManualIndexerAndKistler THEN

                        eProcessCycleState :=
                            E_ProcessCycle_State.WAIT_AFTER_KISTLER;

                    ELSE

                        eProcessCycleState :=
                            E_ProcessCycle_State.IDLE;

                    END_IF

                END_IF

            // =================================================================
            E_ProcessCycle_State.WAIT_AFTER_KISTLER:
            // =================================================================

                IF stKistlerOutTelegram.bSequenceEnd
                   AND
                   (
                       stKistlerOutTelegram.bHomePosReached
                       OR stKistlerOutTelegram.bRefPosReached
                       OR stKistler_Status.bInPosition
                   ) THEN

                    GVL_MASTER.stProcess.bReleaseNestRotation := TRUE;

                    eProcessCycleState :=
                        E_ProcessCycle_State.RELEASE_NEST;

                END_IF

            // =================================================================
            E_ProcessCycle_State.RELEASE_NEST:
            // =================================================================

                GVL_MASTER.stProcess.bReleaseNestRotation := TRUE;

                IF eNestState <> E_NestState.TESTING
                   OR NOT GVL_MASTER.stProcess.bNestTestingReady THEN

                    GVL_MASTER.stProcess.bReleaseNestRotation := FALSE;
                    GVL_MASTER.stProcess.bKistlerCycleRequest := FALSE;
                    GVL_MASTER.stProcess.bKistlerCycleDone := FALSE;
                    GVL_MASTER.stProcess.bKistlerHomeDone := FALSE;

                    tonAfterKistlerDelay(IN := FALSE);

                    IF bManualIndexerOnly
                       OR bManualIndexerAndKistler THEN

                        eProcessCycleState :=
                            E_ProcessCycle_State.WAIT_NEST_TESTING_READY;

                    ELSE

                        eProcessCycleState :=
                            E_ProcessCycle_State.IDLE;

                    END_IF

                END_IF

            // =================================================================
            E_ProcessCycle_State.FAULT:
            // =================================================================

                GVL_MASTER.stProcess.bKistlerCycleRequest := FALSE;
                GVL_MASTER.stProcess.bReleaseNestRotation := FALSE;

                tonAfterKistlerDelay(IN := FALSE);

                M_ResetProcessCycle();

                GVL_MASTER.stMachineStatus.eMachineState :=
                    E_MachineState.FAULT;

            // =================================================================
            ELSE
            // =================================================================

                eProcessCycleState :=
                    E_ProcessCycle_State.IDLE;

        END_CASE

END_CASE

M_ProcessCycle := TRUE;
END_METHOD

METHOD PRIVATE M_PuckLockerDisposition
VAR
	iOperatorNestIndex : INT;
    bResultPass        : BOOL;
    bResultFail        : BOOL;
END_VAR
// -----------------------------------------------------------------------------
// Do not generate dispositions when the Puck Locker is disabled.
// -----------------------------------------------------------------------------
(*IF GVL_HMI.stPuckLocker.eMode = E_PuckLockerMode.Disabled THEN
    RETURN;
END_IF*)


// -----------------------------------------------------------------------------
// The operator nest must be known.
// -----------------------------------------------------------------------------
IF eOperatorNestPosition = E_NestPosition.Unknown THEN
    RETURN;
END_IF


// Process the operator disposition whenever the table is stationary,
// mechanically locked and accessible to the operator.
//
// TESTING:
//     Normal production flow.
//
// WAIT_OPERATOR_EXCHANGE:
//     Normal exchange after a completed test.
//
// IDLE:
//     Recovery flow after FAULT, STOPPED or reinitialisation.
IF (
        eNestState <> E_NestState.IDLE
        AND eNestState <> E_NestState.TESTING
        AND eNestState <> E_NestState.WAIT_OPERATOR_EXCHANGE
   )
   OR GVL_MASTER.stNestTable.bNestInMotion
   OR NOT GVL_MASTER.stNestTable.bNestReadySensor
   OR NOT GVL_MASTER.stNestTable.bNestLockedSensor
   OR eCurrentNestPos = E_NestPosition.Unknown THEN

    RETURN;

END_IF


// -----------------------------------------------------------------------------
// E_NestPosition values correspond directly to array indexes 1..4.
// -----------------------------------------------------------------------------
iOperatorNestIndex := eOperatorNestPosition;

IF (iOperatorNestIndex < 1) OR (iOperatorNestIndex > 4) THEN
    RETURN;
END_IF


// -----------------------------------------------------------------------------
// The nest currently accessible to the operator must contain a valid result.
// -----------------------------------------------------------------------------
IF NOT GVL_MASTER.astNestProcessResult[iOperatorNestIndex].bResultValid THEN
    RETURN;
END_IF


// -----------------------------------------------------------------------------
// Do not process the same nest disposition more than once.
// -----------------------------------------------------------------------------
IF GVL_MASTER.astNestProcessResult[iOperatorNestIndex].bDispositionSent THEN
    RETURN;
END_IF


// -----------------------------------------------------------------------------
// -----------------------------------------------------------------------------
// Copy the result locally for validation and readability.
// -----------------------------------------------------------------------------
bResultPass :=
    GVL_MASTER.astNestProcessResult[iOperatorNestIndex].bPass;

bResultFail :=
    GVL_MASTER.astNestProcessResult[iOperatorNestIndex].bFail;


// -----------------------------------------------------------------------------
// The result must contain exactly one disposition.
//
// Invalid combinations:
//     PASS = FALSE and FAIL = FALSE
//     PASS = TRUE  and FAIL = TRUE
// -----------------------------------------------------------------------------
IF bResultPass = bResultFail THEN
    RETURN;
END_IF


// -----------------------------------------------------------------------------
// PUCK LOCKER DISABLED:
//
// There is no physical locker handshake to perform.
//
// Mark the disposition as delivered internally so that the operator exchange
// sequence can continue using the normal PASS/FAIL result.
//
// FAIL still requires:
//     1. Part removal from the operator nest.
//     2. Confirmation from the reject-bin sensor.
//
// No puck presence or puck locked condition is required.
// -----------------------------------------------------------------------------
IF GVL_HMI.stPuckLocker.eMode = E_PuckLockerMode.Disabled THEN

    GVL_MASTER.astNestProcessResult[
        iOperatorNestIndex
    ].bDispositionSent := TRUE;
    RETURN;
END_IF


// -----------------------------------------------------------------------------
// A previous disposition was already sent and is still waiting for confirmation
// from PRG_PuckLocker.
// -----------------------------------------------------------------------------
IF ePendingPuckDispositionNest <> E_NestPosition.Unknown THEN
    RETURN;
END_IF




// -----------------------------------------------------------------------------
// Do not overwrite a disposition that has not yet been consumed by the locker.
// -----------------------------------------------------------------------------
IF GVL_MASTER.stPuckLocker.bApplyDisposition
   OR GVL_MASTER.stPuckLocker.bDispositionPending THEN

    RETURN;
END_IF


// -----------------------------------------------------------------------------
// PASS:
// Authorise the release of one puck.
// -----------------------------------------------------------------------------
IF bResultPass THEN

    GVL_MASTER.stPuckLocker.nRequestedRelease := 1;
    GVL_MASTER.stPuckLocker.nRequestedRemoval := 0;

    // Store the nest that originated this request so that the confirmation
    // remains associated with the correct nest even if the table moves later.
    ePendingPuckDispositionNest := eOperatorNestPosition;

    // Apply the request only after all associated data has been prepared.
    GVL_MASTER.stPuckLocker.bApplyDisposition := TRUE;

// -----------------------------------------------------------------------------
// FAIL:
// Inform the locker of the rejected result, but do not authorise puck release.
// The puck must remain locked until a future PASS result is received.
// -----------------------------------------------------------------------------
ELSIF bResultFail THEN

    GVL_MASTER.stPuckLocker.nRequestedRelease := 0;
    GVL_MASTER.stPuckLocker.nRequestedRemoval := 1;

    ePendingPuckDispositionNest := eOperatorNestPosition;

    // Apply the request only after all associated data has been prepared.
    GVL_MASTER.stPuckLocker.bApplyDisposition := TRUE;

END_IF
END_METHOD

METHOD PRIVATE M_ResetProcessCycle : BOOL
VAR_INPUT

END_VAR
M_ResetProcessCycle := FALSE;

eProcessCycleState := E_ProcessCycle_State.IDLE;


// =========================================================
// RESET PROCESS FLAGS
// =========================================================

GVL_MASTER.stProcess.bKistlerCycleRequest := FALSE;
GVL_MASTER.stProcess.bKistlerCycleDone := FALSE;
GVL_MASTER.stProcess.bKistlerHomeDone := FALSE;
GVL_MASTER.stProcess.bNestTestingReady := FALSE;
GVL_MASTER.stProcess.bReleaseNestRotation := FALSE;
GVL_MASTER.stProcess.bKistlerResultOK := FALSE;
GVL_MASTER.stProcess.bKistlerResultNOK := FALSE;





// =========================================================
// RESET PROCESS TIMERS
// =========================================================

tonGuideCylinderDelay(IN := FALSE);
tonGuideCylinderRetractDelay(IN := FALSE);
tonAfterKistlerDelay(IN := FALSE);


// =========================================================
// RESET ACTUATOR REQUESTS
// =========================================================

GVL_MASTER.stActuators.bGuideCylinderExtendRequest := FALSE;

GVL_MASTER.stNestTable.bSupportExtendRequest := FALSE;
GVL_MASTER.stNestTable.bSupportRetractRequest := TRUE;


// =========================================================
// RESET HMI MANUAL COMMANDS
// =========================================================

GVL_HMI.i_bHMIManualModeRequest := FALSE;
GVL_HMI.i_bHMIIndexerManualEnable := FALSE;
GVL_HMI.i_bHMIKistlerManualEnable := FALSE;


// =========================================================
// RESET KISTLER SEQUENCE COMMANDS
// =========================================================

stKistler_CMD.bStart := FALSE;
stKistler_CMD.bRunSequence := FALSE;
stKistler_CMD.bDriveToHome := FALSE;
stKistler_CMD.bDriveToRef := FALSE;
stKistler_CMD.bContinueFromWait := FALSE;
stKistler_CMD.bTareY := FALSE;



// =========================================================
// RESET ROUTINE COMPLETE
// =========================================================

M_ResetProcessCycle := TRUE;
END_METHOD

METHOD PRIVATE M_StartFaultRejectRecovery
VAR
    iNestIndex : INT;
END_VAR

// -----------------------------------------------------------------------------
// Start the fault-recovery reject sequence.
//
// The nest that was at the operator position when the fault occurred is
// excluded. The other three physical nests are marked as rejected and will
// later be discarded using the normal operator exchange and reject flow.
// -----------------------------------------------------------------------------

IF eOperatorNestPosition = E_NestPosition.UNKNOWN THEN
    RETURN;
END_IF


// Save the physical nest that was at the operator position.
eFaultOperatorNest := eOperatorNestPosition;


// Preserve the actual Kistler result during fault recovery.
//
// A machine fault is not a Kistler FAIL result.
// The retained nest memory determines the real part state:
//
// bResultValid = TRUE  -> keep the existing PASS / FAIL result.
// bResultValid = FALSE -> part remains NOT TESTED.
//
// This also covers a Kistler cycle interrupted by a machine fault:
// because no valid Kistler result was completed, no artificial
// FAIL result is generated here.
FOR iNestIndex := 1 TO 4 DO

    IF GVL_MASTER.astNestTracking[iNestIndex].bPartLoaded THEN

        GVL_MASTER.astNestProcessResult[
            iNestIndex
        ].bDispositionSent := FALSE;

        // If the part currently at the Kistler station does not have
        // a valid completed result, the test cannot be guaranteed.
        // Treat this part as FAIL for reject handling.
        IF (iNestIndex = TO_INT(eKistlerNestPosition))
           AND NOT GVL_MASTER.astNestProcessResult[iNestIndex].bResultValid THEN

            GVL_MASTER.astNestProcessResult[
                iNestIndex
            ].bResultValid := TRUE;

            GVL_MASTER.astNestProcessResult[
                iNestIndex
            ].bPass := FALSE;

            GVL_MASTER.astNestProcessResult[
                iNestIndex
            ].bFail := TRUE;

            GVL_HMI.aKistlerNestResult[
                iNestIndex
            ].eResult := E_HMIKistlerResult.FAIL;

        END_IF

    END_IF

END_FOR


bFaultRejectPending := TRUE;
bFaultRejectActive := TRUE;
END_METHOD

METHOD PRIVATE M_StatusMapping : BOOL
VAR

tonKistlerWarningFilter	: TON;


END_VAR

// =================================================================================
// KISTLER TO GLOBAL STATUS MAPPING
// =================================================================================
// Link the software/hardware safety loop to the machine status structure
GVL_MASTER.stMachineStatus.bSafety := GVL_IO.stSafety.bSystemSafeOK;

// Map the local Kistler hardware ready flag to our main control variable
bKistlerReady := stKistler_Status.bReady;

// Update the global machine fault status if the Kistler press enters an error state
IF stKistler_Status.bError THEN
	GVL_MASTER.stMachineStatus.bFault := TRUE;
END_IF

// =================================================================================
// HMI / PANEL LAMP SIGNALLING MANAGEMENT
// =================================================================================
// Control the Start Button Lamp feedback based on machine state
IF GVL_MASTER.stMachineStatus.eMachineState = E_MachineState.STOPPED AND bKistlerReady THEN
    GVL_MASTER.bStartButtonLamp := GVL_MASTER.bBlink_1Hz; // Uses standard 1Hz global clock bit
ELSIF GVL_MASTER.stMachineStatus.eMachineState = E_MachineState.SYSTEM_AUTO_CYCLE THEN
    GVL_MASTER.bStartButtonLamp := TRUE;
ELSE
    GVL_MASTER.bStartButtonLamp := FALSE;
END_IF

// =================================================================================
// GLOBAL DIAGNOSTIC MAPPING
// =================================================================================

// Stop request
GVL_MASTER.stDiagnostics.bStopRequested := bStopRequested;

// Machine sequence timeouts
GVL_MASTER.stDiagnostics.bInitialisationTimeout := tonSys_InitTimeout.Q;

GVL_MASTER.stDiagnostics.bProcessTimeout := tonTimeout_testing.Q;

// Main Kistler status
GVL_MASTER.stDiagnostics.bKistlerError := stKistler_Status.bError;

GVL_MASTER.stDiagnostics.bKistlerBusy := stKistler_Status.bBusy;

GVL_MASTER.stDiagnostics.bKistlerNotReady := NOT stKistler_Status.bReady;

// Detailed Kistler telegram diagnostics
GVL_MASTER.stDiagnostics.bKistlerAlarm := stKistlerOutTelegram.bAlarm;

tonKistlerWarningFilter( IN := stKistlerOutTelegram.bWarning, PT := T#3S);
GVL_MASTER.stDiagnostics.bKistlerWarning := tonKistlerWarningFilter.Q;

GVL_MASTER.stDiagnostics.bKistlerSequenceError := stKistlerOutTelegram.bSequenceError;

GVL_MASTER.stDiagnostics.bKistlerServoError := stKistlerOutTelegram.bServoError;

GVL_MASTER.stDiagnostics.bKistlerTransmissionFault := stKistlerOutTelegram.bTransmissionFault;

GVL_MASTER.stDiagnostics.bKistlerDeviceUnavailable := NOT stKistlerOutTelegram.bDeviceAvailable;

// =================================================================================
// Nest-table diagnostics
// =================================================================================

// Recoverable wrong-position condition.
// Active while the nest state machine is in WRONG_POSITION.
GVL_MASTER.stDiagnostics.bNestWrongPositionAlarm := eNestState = E_NestState.WRONG_POSITION;


// Wrong-position fault.
// Active when the recovery timeout has expired.
GVL_MASTER.stDiagnostics.bNestWrongPosition :=  bNestWrongPositionFault;

// =================================================================================
// METHOD EXECUTION FEEDBACK (Return True)
// =================================================================================
// Returning TRUE confirms that the status mapping routine executed successfully
M_StatusMapping := TRUE;
END_METHOD

METHOD M_StoreKistlerResult
VAR
	iNestIndex : INT;
END_VAR
IF eKistlerNestPosition = E_NestPosition.Unknown THEN
    RETURN;
END_IF;

iNestIndex := eKistlerNestPosition;

IF (iNestIndex < 1) OR (iNestIndex > 4) THEN
    RETURN;
END_IF;

// Prevent writing the same result repeatedly for several PLC scans.
IF bKistlerResultStored THEN
    RETURN;
END_IF;

IF stKistler_Status.bPartOK THEN

    GVL_MASTER.astNestProcessResult[iNestIndex].bResultValid := TRUE;
    GVL_MASTER.astNestProcessResult[iNestIndex].bPass := TRUE;
    GVL_MASTER.astNestProcessResult[iNestIndex].bFail := FALSE;
    GVL_MASTER.astNestProcessResult[iNestIndex].bDispositionSent := FALSE;

    bKistlerResultStored := TRUE;

ELSIF stKistler_Status.bPartNOK THEN

    GVL_MASTER.astNestProcessResult[iNestIndex].bResultValid := TRUE;
    GVL_MASTER.astNestProcessResult[iNestIndex].bPass := FALSE;
    GVL_MASTER.astNestProcessResult[iNestIndex].bFail := TRUE;
    GVL_MASTER.astNestProcessResult[iNestIndex].bDispositionSent := FALSE;

    bKistlerResultStored := TRUE;

END_IF;
END_METHOD

METHOD M_SupportControl
VAR_INPUT
    bExtendRequest  : BOOL; // Request to lift support
    bRetractRequest : BOOL; // Request to lower support
END_VAR
// =================================================================
// SUPPORT CYLINDER CONTROL
// =================================================================
// This method is responsible only for the support cylinder outputs.
// It does not decide Auto Cycle or Manual Mode.
// The request must come from M_ProcessCycle, M_NestTableControl,
// or later from the Kistler coordination logic.

// Safety priority: never command both coils at the same time.
IF bExtendRequest AND NOT bRetractRequest THEN

    // Lift support
    GVL_MASTER.stNestTable.qSupportExtend  := TRUE;
    GVL_MASTER.stNestTable.qSupportRetract := FALSE;


ELSIF bRetractRequest AND NOT bExtendRequest THEN

    // Lower support
    GVL_MASTER.stNestTable.qSupportExtend  := FALSE;
    GVL_MASTER.stNestTable.qSupportRetract := TRUE;



ELSE

    // No request or conflicting request:
    // keep both outputs off to avoid fighting the pneumatic valve.
    GVL_MASTER.stNestTable.qSupportExtend  := FALSE;
    GVL_MASTER.stNestTable.qSupportRetract := FALSE;



END_IF
END_METHOD

METHOD PRIVATE M_TerminalInfo
VAR_INPUT
END_VAR
(*
    Updates the diagnostic information for all Beckhoff terminals.

    The terminal state value must already be mapped from the EtherCAT
    terminal diagnostic input to:

        stTerminalInfo.nTerminal_State
*)

GVL_IO.stTerm_Ek1100.stTerminalInfo.fbTerminalInfo(
    nTerminalState         := GVL_IO.stTerm_Ek1100.stTerminalInfo.nTerminal_State,
    sTerminalState         => GVL_IO.stTerm_Ek1100.stTerminalInfo.sTerminalInfo,
    bTerminalOperational   => GVL_IO.stTerm_Ek1100.stTerminalInfo.bTerminalOperational
);

GVL_IO.stTerm2_EL6070.stTerminalInfo.fbTerminalInfo(
    nTerminalState         := GVL_IO.stTerm2_EL6070.stTerminalInfo.nTerminal_State,
    sTerminalState         => GVL_IO.stTerm2_EL6070.stTerminalInfo.sTerminalInfo,
    bTerminalOperational   => GVL_IO.stTerm2_EL6070.stTerminalInfo.bTerminalOperational
);

GVL_IO.stTerm3_EL6910.stTerminalInfo.fbTerminalInfo(
    nTerminalState         := GVL_IO.stTerm3_EL6910.stTerminalInfo.nTerminal_State,
    sTerminalState         => GVL_IO.stTerm3_EL6910.stTerminalInfo.sTerminalInfo,
    bTerminalOperational   => GVL_IO.stTerm3_EL6910.stTerminalInfo.bTerminalOperational
);

GVL_IO.stTerm4_EL1918.stTerminalInfo.fbTerminalInfo(
    nTerminalState         := GVL_IO.stTerm4_EL1918.stTerminalInfo.nTerminal_State,
    sTerminalState         => GVL_IO.stTerm4_EL1918.stTerminalInfo.sTerminalInfo,
    bTerminalOperational   => GVL_IO.stTerm4_EL1918.stTerminalInfo.bTerminalOperational
);

GVL_IO.stTerm5_EL1918.stTerminalInfo.fbTerminalInfo(
    nTerminalState         := GVL_IO.stTerm5_EL1918.stTerminalInfo.nTerminal_State,
    sTerminalState         => GVL_IO.stTerm5_EL1918.stTerminalInfo.sTerminalInfo,
    bTerminalOperational   => GVL_IO.stTerm5_EL1918.stTerminalInfo.bTerminalOperational
);

GVL_IO.stTerm6_EL1918.stTerminalInfo.fbTerminalInfo(
    nTerminalState         := GVL_IO.stTerm6_EL1918.stTerminalInfo.nTerminal_State,
    sTerminalState         => GVL_IO.stTerm6_EL1918.stTerminalInfo.sTerminalInfo,
    bTerminalOperational   => GVL_IO.stTerm6_EL1918.stTerminalInfo.bTerminalOperational
);

GVL_IO.stTerm7_EL2904.stTerminalInfo.fbTerminalInfo(
    nTerminalState         := GVL_IO.stTerm7_EL2904.stTerminalInfo.nTerminal_State,
    sTerminalState         => GVL_IO.stTerm7_EL2904.stTerminalInfo.sTerminalInfo,
    bTerminalOperational   => GVL_IO.stTerm7_EL2904.stTerminalInfo.bTerminalOperational
);

GVL_IO.stTerm8_EL2904.stTerminalInfo.fbTerminalInfo(
    nTerminalState         := GVL_IO.stTerm8_EL2904.stTerminalInfo.nTerminal_State,
    sTerminalState         => GVL_IO.stTerm8_EL2904.stTerminalInfo.sTerminalInfo,
    bTerminalOperational   => GVL_IO.stTerm8_EL2904.stTerminalInfo.bTerminalOperational
);

GVL_IO.stTerm9_EL1809.stTerminalInfo.fbTerminalInfo(
    nTerminalState         := GVL_IO.stTerm9_EL1809.stTerminalInfo.nTerminal_State,
    sTerminalState         => GVL_IO.stTerm9_EL1809.stTerminalInfo.sTerminalInfo,
    bTerminalOperational   => GVL_IO.stTerm9_EL1809.stTerminalInfo.bTerminalOperational
);

GVL_IO.stTerm10_EL1809.stTerminalInfo.fbTerminalInfo(
    nTerminalState         := GVL_IO.stTerm10_EL1809.stTerminalInfo.nTerminal_State,
    sTerminalState         => GVL_IO.stTerm10_EL1809.stTerminalInfo.sTerminalInfo,
    bTerminalOperational   => GVL_IO.stTerm10_EL1809.stTerminalInfo.bTerminalOperational
);

GVL_IO.stTerm11_EL2809.stTerminalInfo.fbTerminalInfo(
    nTerminalState         := GVL_IO.stTerm11_EL2809.stTerminalInfo.nTerminal_State,
    sTerminalState         => GVL_IO.stTerm11_EL2809.stTerminalInfo.sTerminalInfo,
    bTerminalOperational   => GVL_IO.stTerm11_EL2809.stTerminalInfo.bTerminalOperational
);

GVL_IO.stTerm12_EL9410.stTerminalInfo.fbTerminalInfo(
    nTerminalState         := GVL_IO.stTerm12_EL9410.stTerminalInfo.nTerminal_State,
    sTerminalState         => GVL_IO.stTerm12_EL9410.stTerminalInfo.sTerminalInfo,
    bTerminalOperational   => GVL_IO.stTerm12_EL9410.stTerminalInfo.bTerminalOperational
);

GVL_IO.stTerm13_EL2809.stTerminalInfo.fbTerminalInfo(
    nTerminalState         := GVL_IO.stTerm13_EL2809.stTerminalInfo.nTerminal_State,
    sTerminalState         => GVL_IO.stTerm13_EL2809.stTerminalInfo.sTerminalInfo,
    bTerminalOperational   => GVL_IO.stTerm13_EL2809.stTerminalInfo.bTerminalOperational
);

GVL_IO.stTerm14_EL3058.stTerminalInfo.fbTerminalInfo(
    nTerminalState         := GVL_IO.stTerm14_EL3058.stTerminalInfo.nTerminal_State,
    sTerminalState         => GVL_IO.stTerm14_EL3058.stTerminalInfo.sTerminalInfo,
    bTerminalOperational   => GVL_IO.stTerm14_EL3058.stTerminalInfo.bTerminalOperational
);

// -----------------------------------------------------------------------------
// T04 - EL1918 channel mirrors for HMI diagnostics
// -----------------------------------------------------------------------------
GVL_IO.stSafety.bEStopCH1 := GVL_IO.stTerm4_EL1918.iEL1918_Ch1;
GVL_IO.stSafety.bEStopCH2 := GVL_IO.stTerm4_EL1918.iEL1918_Ch2;
GVL_MASTER.i_bButtonReset := GVL_IO.stTerm4_EL1918.iEL1918_Ch3;

// -----------------------------------------------------------------------------
// T05 - EL1918 channel mirrors for HMI diagnostics
// -----------------------------------------------------------------------------

GVL_IO.stSafety.bTwoHandsLeft := GVL_IO.stTerm5_EL1918.iEL1918_Ch3;
GVL_IO.stSafety.bTwoHandsRight := GVL_IO.stTerm5_EL1918.iEL1918_Ch4;

// -----------------------------------------------------------------------------
// T06 - EL1918 channel mirrors for HMI diagnostics
// -----------------------------------------------------------------------------

GVL_IO.stSafety.bDoorFlapLeftCH1  := GVL_IO.stTerm6_EL1918.iEL1918_Ch1;
GVL_IO.stSafety.bDoorFlapLeftCH2  := GVL_IO.stTerm6_EL1918.iEL1918_Ch2;
GVL_IO.stSafety.bDoorFlapRightCH1 := GVL_IO.stTerm6_EL1918.iEL1918_Ch4;
GVL_IO.stSafety.bDoorFlapRightCH2 := GVL_IO.stTerm6_EL1918.iEL1918_Ch5;
// -----------------------------------------------------------------------------
// T07- EL2904 channel mirrors for HMI diagnostics
// -----------------------------------------------------------------------------
GVL_IO.stTerm7_EL2904.qEL2904_Ch1 := GVL_IO.stSafety.bAirSupplyEnabled;
GVL_IO.stTerm7_EL2904.qEL2904_Ch2 := GVL_IO.stSafety.bSafetyReset;
GVL_IO.stTerm7_EL2904.qEL2904_Ch3 := GVL_IO.stSafety.bMainDoorLocked;
GVL_IO.stTerm7_EL2904.qEL2904_Ch4 := FALSE;

// -----------------------------------------------------------------------------
// T08- EL2904 channel mirrors for HMI diagnostics
// -----------------------------------------------------------------------------
GVL_IO.stTerm8_EL2904.qEL2904_Ch1 := GVL_IO.stSafety.bSafetyRelayIndraDrive;
GVL_IO.stTerm8_EL2904.qEL2904_Ch2 := GVL_IO.stSafety.bIndraDriveEStop;
GVL_IO.stTerm8_EL2904.qEL2904_Ch3 := GVL_IO.stSafety.bSafetyRelayEStop;
GVL_IO.stTerm8_EL2904.qEL2904_Ch4 := FALSE;
// -----------------------------------------------------------------------------
// T09 - EL1809 channel mirrors for HMI diagnostics
// -----------------------------------------------------------------------------
GVL_MASTER.i_bButtonStart 							:= GVL_IO.stTerm9_EL1809.iEL1809_Ch1;
GVL_MASTER.i_bButtonStop 							:= GVL_IO.stTerm9_EL1809.iEL1809_Ch2;
GVL_MASTER.bUp24VPowerSupplyOk 						:= GVL_IO.stTerm9_EL1809.iEL1809_Ch3;
GVL_MASTER.bUs24VPowerSupplyOk 						:= GVL_IO.stTerm9_EL1809.iEL1809_Ch4;
GVL_MASTER.stSensors.bPartPresent_Reject 			:= GVL_IO.stTerm9_EL1809.iEL1809_Ch5;
GVL_MASTER.stNestTable.bNestPos_1_Sensor 			:= GVL_IO.stTerm9_EL1809.iEL1809_Ch6;
GVL_MASTER.stNestTable.bNestPos_2_Sensor 			:= GVL_IO.stTerm9_EL1809.iEL1809_Ch7;
GVL_MASTER.stNestTable.bNestPos_3_Sensor 			:= GVL_IO.stTerm9_EL1809.iEL1809_Ch8;
GVL_MASTER.stNestTable.bNestCompletedSensor 		:= GVL_IO.stTerm9_EL1809.iEL1809_Ch9;
GVL_MASTER.stNestTable.bNestLockedSensor 			:= GVL_IO.stTerm9_EL1809.iEL1809_Ch10;
GVL_MASTER.stNestTable.bNestReadySensor 			:= GVL_IO.stTerm9_EL1809.iEL1809_Ch11;
GVL_MASTER.stSensors.bPartPresent_NEST 				:= GVL_IO.stTerm9_EL1809.iEL1809_Ch12;
GVL_MASTER.stSensors.bPartPresent_Kistler 			:= GVL_IO.stTerm9_EL1809.iEL1809_Ch13;

// -----------------------------------------------------------------------------
// T10 - EL1809 channel mirrors for HMI diagnostics
// -----------------------------------------------------------------------------
GVL_MASTER.stNestTable.bSupportRetracted := GVL_IO.stTerm10_EL1809.iEL1809_Ch1;
GVL_MASTER.stNestTable.bSupportExtended := GVL_IO.stTerm10_EL1809.iEL1809_Ch2;
// -----------------------------------------------------------------------------
// T11 - EL12809 channel mirrors for HMI diagnostics
// -----------------------------------------------------------------------------

GVL_IO.stTerm11_EL2809.iEL2809_Ch1 := PRG_MachineControl.q_bLED_Start;
GVL_IO.stTerm11_EL2809.iEL2809_Ch2 := PRG_MachineControl.q_bLED_Reset;
GVL_IO.stTerm11_EL2809.iEL2809_Ch3 := PRG_MachineControl.q_bLED_Fail;
GVL_IO.stTerm11_EL2809.iEL2809_Ch4 := PRG_MachineControl.q_bLED_Pass;
GVL_IO.stTerm11_EL2809.iEL2809_Ch5 := GVL_IO.qInternalLight;
GVL_IO.stTerm11_EL2809.iEL2809_Ch6 := GVL_MASTER.stNestTable.qNestRotatePortB;
GVL_IO.stTerm11_EL2809.iEL2809_Ch7 := GVL_MASTER.stNestTable.qNestRotatePortA;
GVL_IO.stTerm11_EL2809.iEL2809_Ch8 := GVL_MASTER.stNestTable.qSupportExtend;
GVL_IO.stTerm11_EL2809.iEL2809_Ch9 := GVL_MASTER.stNestTable.qSupportRetract;
GVL_IO.stTerm11_EL2809.iEL2809_Ch10 := GVL_MASTER.stActuators.qGuideCylinder;
GVL_IO.stTerm11_EL2809.iEL2809_Ch11 := FALSE;
GVL_IO.stTerm11_EL2809.iEL2809_Ch12 := FALSE;
GVL_IO.stTerm11_EL2809.iEL2809_Ch13 := FALSE;
GVL_IO.stTerm11_EL2809.iEL2809_Ch14 := FALSE;
GVL_IO.stTerm11_EL2809.iEL2809_Ch15 := FALSE;
GVL_IO.stTerm11_EL2809.iEL2809_Ch16 := FALSE;


// -----------------------------------------------------------------------------
// T13 - EL12809 channel mirrors for HMI diagnostics
// -----------------------------------------------------------------------------

GVL_IO.stTerm13_EL2809.iEL2809_Ch9 := GVL_IO.qExternalLight;
END_METHOD

METHOD PRIVATE M_UpdateActiveNestPositions
VAR_INPUT
END_VAR
eKistlerNestPosition := eCurrentNestPos;

eOperatorNestPosition := F_GetOppositeNestPosition( eKistlerPosition := eKistlerNestPosition );

IF eKistlerNestPosition <> E_NestPosition.Unknown THEN

    iKistlerNestIndex := TO_INT(eKistlerNestPosition);

ELSE

    iKistlerNestIndex := 0;

END_IF;

IF eOperatorNestPosition <> E_NestPosition.Unknown THEN

    iOperatorNestIndex := TO_INT(eOperatorNestPosition);

ELSE

    iOperatorNestIndex := 0;

END_IF;
END_METHOD

METHOD PRIVATE M_UpdateMachineMessage
VAR
	bPuckLockerEnabled	: BOOL;
END_VAR
// -----------------------------------------------------------------------------
// Default message.
// -----------------------------------------------------------------------------
sMachineMessage := '';

bPuckLockerEnabled :=
    GVL_HMI.stPuckLocker.eMode <>
        E_PuckLockerMode.Disabled;


// -----------------------------------------------------------------------------
// Machine messages are currently used during Automatic Cycle.
// -----------------------------------------------------------------------------

IF GVL_MASTER.stMachineStatus.eMachineState =
    E_MachineState.SYSTEM_AUTO_CYCLE THEN


    // =========================================================================
    // Highest priority:
    // Index table stopped in a recoverable wrong position.
    // =========================================================================
    IF GVL_MASTER.stDiagnostics.bNestWrongPositionAlarm THEN

        sMachineMessage :=
            'Index wrong position - place both hands on the safety controls to recover';


    // =========================================================================
    // Second priority:
    // The table is physically moving.
    // =========================================================================
    ELSIF GVL_MASTER.stNestTable.bNestInMotion THEN

        sMachineMessage :=
            'Index table moving - keep hands clear';


    ELSE

        // =====================================================================
        // Operator-exchange sequence.
        //
        // Messages follow the exact same state machine that controls table
        // permission. This prevents instructions from appearing out of order.
        // =====================================================================

        CASE eOperatorExchangeState OF


            // =================================================================
            E_OperatorExchangeState.Idle:
            // =================================================================

                IF bPuckLockerEnabled THEN

                    // ---------------------------------------------------------
                    // Puck Locker enabled:
                    // first require the puck to be present and locked.
                    // ---------------------------------------------------------
                    IF NOT GVL_MASTER.stPuckLocker.bPuckDetected THEN

                        sMachineMessage :=
                            'Insert puck into locker to continue';

                    ELSIF
                        NOT GVL_MASTER.stPuckLocker.bPuckLocked
                        OR
                        GVL_MASTER.stPuckLocker.eState <>
                            E_PuckLockerState.Locked THEN

                        sMachineMessage :=
                            'Waiting for puck locker to lock';

                    ELSIF NOT GVL_MASTER.stSensors.bPartPresent_NEST THEN

                        sMachineMessage :=
                            'Load part into operator nest';

                    ELSE

                        sMachineMessage :=
                            'Ready to index - press both safety controls';

                    END_IF


                ELSE

                    // ---------------------------------------------------------
                    // Puck Locker disabled:
                    // an empty operator nest is allowed to continue.
                    // ---------------------------------------------------------
                    IF GVL_MASTER.stSensors.bPartPresent_NEST THEN

                        sMachineMessage :=
                            'Part loaded - press both safety controls to index';

                    ELSE

                        sMachineMessage :=
                            'Load new part or press both safety controls to continue';

                    END_IF

                END_IF


            // =================================================================
            E_OperatorExchangeState.WaitingForPartRemoval:
            // =================================================================

                // The processed part must always be removed first.
                IF bPendingOperatorResultFail THEN

                    sMachineMessage :=
                        'Remove failed part from operator nest';

